DATA_BLOCK "coordinate"	// DB 22
VERSION : 0.1
  STRUCT
   CoordSaldaturaPP1 : ARRAY  [1 .. 20 ] OF //Coordinates of points
   STRUCT
    X1 : DINT ;	//X coordinate of point PP1
    Y1 : DINT ;	//Y coordinate of point PP1
    X2 : DINT ;
    Y2 : DINT ;
   END_STRUCT ;
   CoordSaldaturaPP2 : ARRAY  [1 .. 20 ] OF //Coordinates of points
   STRUCT
    X1 : DINT ;	//X coordinate of point PP2
    Y1 : DINT ;	//Y coordinate of point PP2
    X2 : DINT ;
    Y2 : DINT ;
   END_STRUCT ;
   CoordSaldaturaPP3 : ARRAY  [1 .. 20 ] OF //Coordinates of points
   STRUCT
    X1 : DINT ;	//X coordinate of point PP3
    Y1 : DINT ;	//Y coordinate of point PP3
    X2 : DINT ;
    Y2 : DINT ;
   END_STRUCT ;
   CoordSaldaturaPP4 : ARRAY  [1 .. 20 ] OF //Coordinates of points
   STRUCT
    X1 : DINT ;	//X coordinate of point PP4
    Y1 : DINT ;	//Y coordinate of point PP4
    X2 : DINT ;
    Y2 : DINT ;
   END_STRUCT ;
   CoordSaldaturaPP5 : ARRAY  [1 .. 20 ] OF //Coordinates of points
   STRUCT
    X1 : DINT ;	//X coordinate of point PP5
    Y1 : DINT ;	//Y coordinate of point PP5
    X2 : DINT ;
    Y2 : DINT ;
   END_STRUCT ;
   CoordSaldaturaPP6 : ARRAY  [1 .. 20 ] OF STRUCT
    X1 : DINT ;
    Y1 : DINT ;
    X2 : DINT ;
    Y2 : DINT ;
   END_STRUCT ;
   CoordSaldaturaPP7 : ARRAY  [1 .. 20 ] OF STRUCT
    X1 : DINT ;
    Y1 : DINT ;
    X2 : DINT ;
    Y2 : DINT ;
   END_STRUCT ;
   CoordSaldaturaPP8 : ARRAY  [1 .. 20 ] OF STRUCT
    X1 : DINT ;
    Y1 : DINT ;
    X2 : DINT ;
    Y2 : DINT ;
   END_STRUCT ;
   CoordSaldaturaPP9 : ARRAY  [1 .. 20 ] OF STRUCT
    X1 : DINT ;
    Y1 : DINT ;
    X2 : DINT ;
    Y2 : DINT ;
   END_STRUCT ;
   CoordSaldaturaPP10 : ARRAY  [1 .. 20 ] OF STRUCT
    X1 : DINT ;
    Y1 : DINT ;
    X2 : DINT ;
    Y2 : DINT ;
   END_STRUCT ;
   CoordSaldaturaPP11 : ARRAY  [1 .. 20 ] OF STRUCT
    X1 : DINT ;
    Y1 : DINT ;
    X2 : DINT ;
    Y2 : DINT ;
   END_STRUCT ;
   CoordSaldaturaPP12 : ARRAY  [1 .. 20 ] OF STRUCT
    X1 : DINT ;
    Y1 : DINT ;
    X2 : DINT ;
    Y2 : DINT ;
   END_STRUCT ;
   CoordSaldaturaPP13 : ARRAY  [1 .. 20 ] OF STRUCT
    X1 : DINT ;
    Y1 : DINT ;
    X2 : DINT ;
    Y2 : DINT ;
   END_STRUCT ;
   CoordSaldaturaPP14 : ARRAY  [1 .. 20 ] OF STRUCT
    X1 : DINT ;
    Y1 : DINT ;
    X2 : DINT ;
    Y2 : DINT ;
   END_STRUCT ;
   CoordSaldaturaPP15 : ARRAY  [1 .. 20 ] OF STRUCT
    X1 : DINT ;
    Y1 : DINT ;
    X2 : DINT ;
    Y2 : DINT ;
   END_STRUCT ;
   CoordSaldaturaPP16 : ARRAY  [1 .. 20 ] OF STRUCT
    X1 : DINT ;
    Y1 : DINT ;
    X2 : DINT ;
    Y2 : DINT ;
   END_STRUCT ;
   CoordSaldaturaPP17 : ARRAY  [1 .. 20 ] OF STRUCT
    X1 : DINT ;
    Y1 : DINT ;
    X2 : DINT ;
    Y2 : DINT ;
   END_STRUCT ;
   CoordSaldaturaPP18 : ARRAY  [1 .. 20 ] OF STRUCT
    X1 : DINT ;
    Y1 : DINT ;
    X2 : DINT ;
    Y2 : DINT ;
   END_STRUCT ;
   CoordSaldaturaPP19 : ARRAY  [1 .. 20 ] OF STRUCT
    X1 : DINT ;
    Y1 : DINT ;
    X2 : DINT ;
    Y2 : DINT ;
   END_STRUCT ;
   CoordSaldaturaPP20 : ARRAY  [1 .. 20 ] OF STRUCT
    X1 : DINT ;
    Y1 : DINT ;
    X2 : DINT ;
    Y2 : DINT ;
   END_STRUCT ;
   CoordinateCam_PP1 : ARRAY  [1 .. 10 ] OF STRUCT
    X : DINT ;	//X coordinate of point cam PP1
    Y : DINT ;	//X coordinate of point cam PP1
   END_STRUCT ;
   CoordinateCam_PP2 : ARRAY  [1 .. 10 ] OF STRUCT
    X : DINT ;	//X coordinate of point cam PP1
    Y : DINT ;	//X coordinate of point cam PP1
   END_STRUCT ;
   CoordinateCam_PP3 : ARRAY  [1 .. 10 ] OF STRUCT
    X : DINT ;	//X coordinate of point cam PP1
    Y : DINT ;	//X coordinate of point cam PP1
   END_STRUCT ;
   CoordinateCam_PP4 : ARRAY  [1 .. 10 ] OF STRUCT
    X : DINT ;	//X coordinate of point cam PP1
    Y : DINT ;	//X coordinate of point cam PP1
   END_STRUCT ;
   CoordinateCam_PP5 : ARRAY  [1 .. 10 ] OF STRUCT
    X : DINT ;	//X coordinate of point cam PP1
    Y : DINT ;	//X coordinate of point cam PP1
   END_STRUCT ;
   CoordinateCam_PP6 : ARRAY  [1 .. 10 ] OF STRUCT
    X : DINT ;	//X coordinate of point cam PP1
    Y : DINT ;	//X coordinate of point cam PP1
   END_STRUCT ;
   CoordinateCam_PP7 : ARRAY  [1 .. 10 ] OF STRUCT
    X : DINT ;	//X coordinate of point cam PP1
    Y : DINT ;	//X coordinate of point cam PP1
   END_STRUCT ;
   CoordinateCam_PP8 : ARRAY  [1 .. 10 ] OF STRUCT
    X : DINT ;	//X coordinate of point cam PP1
    Y : DINT ;	//X coordinate of point cam PP1
   END_STRUCT ;
   CoordinateCam_PP9 : ARRAY  [1 .. 10 ] OF STRUCT
    X : DINT ;	//X coordinate of point cam PP1
    Y : DINT ;	//X coordinate of point cam PP1
   END_STRUCT ;
   CoordinateCam_PP10 : ARRAY  [1 .. 10 ] OF STRUCT
    X : DINT ;	//X coordinate of point cam PP1
    Y : DINT ;	//X coordinate of point cam PP1
   END_STRUCT ;
   CoordinateCam_PP11 : ARRAY  [1 .. 10 ] OF STRUCT
    X : DINT ;	//X coordinate of point cam PP1
    Y : DINT ;	//X coordinate of point cam PP1
   END_STRUCT ;
   CoordinateCam_PP12 : ARRAY  [1 .. 10 ] OF STRUCT
    X : DINT ;	//X coordinate of point cam PP1
    Y : DINT ;	//X coordinate of point cam PP1
   END_STRUCT ;
   CoordinateCam_PP13 : ARRAY  [1 .. 10 ] OF STRUCT
    X : DINT ;	//X coordinate of point cam PP1
    Y : DINT ;	//X coordinate of point cam PP1
   END_STRUCT ;
   CoordinateCam_PP14 : ARRAY  [1 .. 10 ] OF STRUCT
    X : DINT ;	//X coordinate of point cam PP1
    Y : DINT ;	//X coordinate of point cam PP1
   END_STRUCT ;
   CoordinateCam_PP15 : ARRAY  [1 .. 10 ] OF STRUCT
    X : DINT ;	//X coordinate of point cam PP1
    Y : DINT ;	//X coordinate of point cam PP1
   END_STRUCT ;
   CoordinateCam_PP16 : ARRAY  [1 .. 10 ] OF STRUCT
    X : DINT ;	//X coordinate of point cam PP1
    Y : DINT ;	//X coordinate of point cam PP1
   END_STRUCT ;
   CoordinateCam_PP17 : ARRAY  [1 .. 10 ] OF STRUCT
    X : DINT ;	//X coordinate of point cam PP1
    Y : DINT ;	//X coordinate of point cam PP1
   END_STRUCT ;
   CoordinateCam_PP18 : ARRAY  [1 .. 10 ] OF STRUCT
    X : DINT ;	//X coordinate of point cam PP1
    Y : DINT ;	//X coordinate of point cam PP1
   END_STRUCT ;
   CoordinateCam_PP19 : ARRAY  [1 .. 10 ] OF STRUCT
    X : DINT ;	//X coordinate of point cam PP1
    Y : DINT ;	//X coordinate of point cam PP1
   END_STRUCT ;
   CoordinateCam_PP20 : ARRAY  [1 .. 10 ] OF STRUCT
    X : DINT ;	//X coordinate of point cam PP1
    Y : DINT ;	//X coordinate of point cam PP1
   END_STRUCT ;
   NumeroSaldaturePP1 : INT ;
   NumeroSaldaturePP2 : INT ;
   NumeroSaldaturePP3 : INT ;
   NumeroSaldaturePP4 : INT ;
   NumeroSaldaturePP5 : INT ;
   NumeroSaldaturePP6 : INT ;
   NumeroSaldaturePP7 : INT ;
   NumeroSaldaturePP8 : INT ;
   NumeroSaldaturePP9 : INT ;
   NumeroSaldaturePP10 : INT ;
   NumeroSaldaturePP11 : INT ;
   NumeroSaldaturePP12 : INT ;
   NumeroSaldaturePP13 : INT ;
   NumeroSaldaturePP14 : INT ;
   NumeroSaldaturePP15 : INT ;
   NumeroSaldaturePP16 : INT ;
   NumeroSaldaturePP17 : INT ;
   NumeroSaldaturePP18 : INT ;
   NumeroSaldaturePP19 : INT ;
   NumeroSaldaturePP20 : INT ;
   TimeWeldingPP1 : ARRAY  [1 .. 20 ] OF STRUCT
    Tempo : S5TIME  := S5T#1S;
   END_STRUCT ;
   TimeWeldingPP2 : ARRAY  [1 .. 20 ] OF STRUCT
    Tempo : S5TIME  := S5T#1S;
   END_STRUCT ;
   TimeWeldingPP3 : ARRAY  [1 .. 20 ] OF STRUCT
    Tempo : S5TIME  := S5T#1S;
   END_STRUCT ;
   TimeWeldingPP4 : ARRAY  [1 .. 20 ] OF STRUCT
    Tempo : S5TIME  := S5T#1S;
   END_STRUCT ;
   TimeWeldingPP5 : ARRAY  [1 .. 20 ] OF STRUCT
    Tempo : S5TIME  := S5T#1S;
   END_STRUCT ;
   TimeWeldingPP6 : ARRAY  [1 .. 20 ] OF STRUCT
    Tempo : S5TIME  := S5T#1S;
   END_STRUCT ;
   TimeWeldingPP7 : ARRAY  [1 .. 20 ] OF STRUCT
    Tempo : S5TIME  := S5T#1S;
   END_STRUCT ;
   TimeWeldingPP8 : ARRAY  [1 .. 20 ] OF STRUCT
    Tempo : S5TIME  := S5T#1S;
   END_STRUCT ;
   TimeWeldingPP9 : ARRAY  [1 .. 20 ] OF STRUCT
    Tempo : S5TIME  := S5T#1S;
   END_STRUCT ;
   TimeWeldingPP10 : ARRAY  [1 .. 20 ] OF STRUCT
    Tempo : S5TIME  := S5T#1S;
   END_STRUCT ;
   TimeWeldingPP11 : ARRAY  [1 .. 20 ] OF STRUCT
    Tempo : S5TIME  := S5T#1S;
   END_STRUCT ;
   TimeWeldingPP12 : ARRAY  [1 .. 20 ] OF STRUCT
    Tempo : S5TIME  := S5T#1S;
   END_STRUCT ;
   TimeWeldingPP13 : ARRAY  [1 .. 20 ] OF STRUCT
    Tempo : S5TIME  := S5T#1S;
   END_STRUCT ;
   TimeWeldingPP14 : ARRAY  [1 .. 20 ] OF STRUCT
    Tempo : S5TIME  := S5T#1S;
   END_STRUCT ;
   TimeWeldingPP15 : ARRAY  [1 .. 20 ] OF STRUCT
    Tempo : S5TIME  := S5T#1S;
   END_STRUCT ;
   TimeWeldingPP16 : ARRAY  [1 .. 20 ] OF STRUCT
    Tempo : S5TIME  := S5T#1S;
   END_STRUCT ;
   TimeWeldingPP17 : ARRAY  [1 .. 20 ] OF STRUCT
    Tempo : S5TIME  := S5T#1S;
   END_STRUCT ;
   TimeWeldingPP18 : ARRAY  [1 .. 20 ] OF STRUCT
    Tempo : S5TIME  := S5T#1S;
   END_STRUCT ;
   TimeWeldingPP19 : ARRAY  [1 .. 20 ] OF STRUCT
    Tempo : S5TIME  := S5T#1S;
   END_STRUCT ;
   TimeWeldingPP20 : ARRAY  [1 .. 20 ] OF STRUCT
    Tempo : S5TIME  := S5T#1S;
   END_STRUCT ;
  END_STRUCT ;	
BEGIN
   CoordSaldaturaPP1[1].X1 := L#-60530;
   CoordSaldaturaPP1[1].Y1 := L#-172340;
   CoordSaldaturaPP1[1].X2 := L#-60530;
   CoordSaldaturaPP1[1].Y2 := L#-172340;
   CoordSaldaturaPP1[2].X1 := L#-46530;
   CoordSaldaturaPP1[2].Y1 := L#-162870;
   CoordSaldaturaPP1[2].X2 := L#-46530;
   CoordSaldaturaPP1[2].Y2 := L#-162870;
   CoordSaldaturaPP1[3].X1 := L#-29630;
   CoordSaldaturaPP1[3].Y1 := L#-163440;
   CoordSaldaturaPP1[3].X2 := L#-29630;
   CoordSaldaturaPP1[3].Y2 := L#-163440;
   CoordSaldaturaPP1[4].X1 := L#-16300;
   CoordSaldaturaPP1[4].Y1 := L#-173820;
   CoordSaldaturaPP1[4].X2 := L#-16300;
   CoordSaldaturaPP1[4].Y2 := L#-173820;
   CoordSaldaturaPP1[5].X1 := L#-11620;
   CoordSaldaturaPP1[5].Y1 := L#-190070;
   CoordSaldaturaPP1[5].X2 := L#-11620;
   CoordSaldaturaPP1[5].Y2 := L#-190070;
   CoordSaldaturaPP1[6].X1 := L#-17370;
   CoordSaldaturaPP1[6].Y1 := L#-205960;
   CoordSaldaturaPP1[6].X2 := L#-17370;
   CoordSaldaturaPP1[6].Y2 := L#-205960;
   CoordSaldaturaPP1[7].X1 := L#-31370;
   CoordSaldaturaPP1[7].Y1 := L#-215430;
   CoordSaldaturaPP1[7].X2 := L#-31370;
   CoordSaldaturaPP1[7].Y2 := L#-215430;
   CoordSaldaturaPP1[8].X1 := L#-48270;
   CoordSaldaturaPP1[8].Y1 := L#-214860;
   CoordSaldaturaPP1[8].X2 := L#-48270;
   CoordSaldaturaPP1[8].Y2 := L#-214860;
   CoordSaldaturaPP1[9].X1 := L#-61600;
   CoordSaldaturaPP1[9].Y1 := L#-204480;
   CoordSaldaturaPP1[9].X2 := L#-61600;
   CoordSaldaturaPP1[9].Y2 := L#-204480;
   CoordSaldaturaPP1[10].X1 := L#-66280;
   CoordSaldaturaPP1[10].Y1 := L#-188230;
   CoordSaldaturaPP1[10].X2 := L#-66280;
   CoordSaldaturaPP1[10].Y2 := L#-188230;
   CoordSaldaturaPP6[1].X1 := L#-24431;
   CoordSaldaturaPP6[1].Y1 := L#-211667;
   CoordSaldaturaPP6[1].X2 := L#-24468;
   CoordSaldaturaPP6[1].Y2 := L#-211634;
   CoordSaldaturaPP6[2].X1 := L#-13011;
   CoordSaldaturaPP6[2].Y1 := L#-199436;
   CoordSaldaturaPP6[2].X2 := L#-12856;
   CoordSaldaturaPP6[2].Y2 := L#-199488;
   CoordSaldaturaPP6[3].X1 := L#-9745;
   CoordSaldaturaPP6[3].Y1 := L#-183598;
   CoordSaldaturaPP6[3].X2 := L#-9756;
   CoordSaldaturaPP6[3].Y2 := L#-183663;
   CoordSaldaturaPP6[4].X1 := L#-16203;
   CoordSaldaturaPP6[4].Y1 := L#-168150;
   CoordSaldaturaPP6[4].X2 := L#-16141;
   CoordSaldaturaPP6[4].Y2 := L#-168156;
   CoordSaldaturaPP6[5].X1 := L#-29434;
   CoordSaldaturaPP6[5].Y1 := L#-158429;
   CoordSaldaturaPP6[5].X2 := L#-29472;
   CoordSaldaturaPP6[5].Y2 := L#-158489;
   CoordSaldaturaPP6[6].X1 := L#-46262;
   CoordSaldaturaPP6[6].Y1 := L#-157658;
   CoordSaldaturaPP6[6].X2 := L#-46155;
   CoordSaldaturaPP6[6].Y2 := L#-157716;
   CoordSaldaturaPP6[7].X1 := L#-60740;
   CoordSaldaturaPP6[7].Y1 := L#-166127;
   CoordSaldaturaPP6[7].X2 := L#-60564;
   CoordSaldaturaPP6[7].Y2 := L#-166296;
   CoordSaldaturaPP6[8].X1 := L#-68335;
   CoordSaldaturaPP6[8].Y1 := L#-180765;
   CoordSaldaturaPP6[8].X2 := L#-68026;
   CoordSaldaturaPP6[8].Y2 := L#-180787;
   CoordSaldaturaPP6[9].X1 := L#-66468;
   CoordSaldaturaPP6[9].Y1 := L#-197254;
   CoordSaldaturaPP6[9].X2 := L#-66217;
   CoordSaldaturaPP6[9].Y2 := L#-197398;
   CoordSaldaturaPP6[10].X1 := L#-56162;
   CoordSaldaturaPP6[10].Y1 := L#-210332;
   CoordSaldaturaPP6[10].X2 := L#-56200;
   CoordSaldaturaPP6[10].Y2 := L#-210331;
   CoordSaldaturaPP6[11].X1 := L#-40981;
   CoordSaldaturaPP6[11].Y1 := L#-215911;
   CoordSaldaturaPP6[11].X2 := L#-40587;
   CoordSaldaturaPP6[11].Y2 := L#-215681;
   CoordSaldaturaPP11[1].X1 := L#-24431;
   CoordSaldaturaPP11[1].Y1 := L#-211667;
   CoordSaldaturaPP11[1].X2 := L#-24468;
   CoordSaldaturaPP11[1].Y2 := L#-211634;
   CoordSaldaturaPP11[2].X1 := L#-13011;
   CoordSaldaturaPP11[2].Y1 := L#-199436;
   CoordSaldaturaPP11[2].X2 := L#-12856;
   CoordSaldaturaPP11[2].Y2 := L#-199488;
   CoordSaldaturaPP11[3].X1 := L#-9745;
   CoordSaldaturaPP11[3].Y1 := L#-183598;
   CoordSaldaturaPP11[3].X2 := L#-9786;
   CoordSaldaturaPP11[3].Y2 := L#-183663;
   CoordSaldaturaPP11[4].X1 := L#-16203;
   CoordSaldaturaPP11[4].Y1 := L#-168150;
   CoordSaldaturaPP11[4].X2 := L#-16141;
   CoordSaldaturaPP11[4].Y2 := L#-168156;
   CoordSaldaturaPP11[5].X1 := L#-29434;
   CoordSaldaturaPP11[5].Y1 := L#-158429;
   CoordSaldaturaPP11[5].X2 := L#-29472;
   CoordSaldaturaPP11[5].Y2 := L#-158489;
   CoordSaldaturaPP11[6].X1 := L#-46262;
   CoordSaldaturaPP11[6].Y1 := L#-157658;
   CoordSaldaturaPP11[6].X2 := L#-46155;
   CoordSaldaturaPP11[6].Y2 := L#-157716;
   CoordSaldaturaPP11[7].X1 := L#-60740;
   CoordSaldaturaPP11[7].Y1 := L#-166127;
   CoordSaldaturaPP11[7].X2 := L#-60564;
   CoordSaldaturaPP11[7].Y2 := L#-166296;
   CoordSaldaturaPP11[8].X1 := L#-68335;
   CoordSaldaturaPP11[8].Y1 := L#-180765;
   CoordSaldaturaPP11[8].X2 := L#-68026;
   CoordSaldaturaPP11[8].Y2 := L#-180787;
   CoordSaldaturaPP11[9].X1 := L#-66468;
   CoordSaldaturaPP11[9].Y1 := L#-197254;
   CoordSaldaturaPP11[9].X2 := L#-66217;
   CoordSaldaturaPP11[9].Y2 := L#-197398;
   CoordSaldaturaPP11[10].X1 := L#-56162;
   CoordSaldaturaPP11[10].Y1 := L#-210332;
   CoordSaldaturaPP11[10].X2 := L#-56200;
   CoordSaldaturaPP11[10].Y2 := L#-210331;
   CoordSaldaturaPP11[11].X1 := L#-40981;
   CoordSaldaturaPP11[11].Y1 := L#-215911;
   CoordSaldaturaPP11[11].X2 := L#-40587;
   CoordSaldaturaPP11[11].Y2 := L#-215681;
   CoordinateCam_PP1[1].X := L#7915;
   CoordinateCam_PP1[1].Y := L#-68282;
   NumeroSaldaturePP1 := 10;
   TimeWeldingPP1[1].Tempo := S5T#1S;
   TimeWeldingPP1[2].Tempo := S5T#2S;
   TimeWeldingPP1[3].Tempo := S5T#1S;
   TimeWeldingPP1[4].Tempo := S5T#1S;
   TimeWeldingPP1[5].Tempo := S5T#1S;
   TimeWeldingPP1[6].Tempo := S5T#1S;
   TimeWeldingPP1[7].Tempo := S5T#1S;
   TimeWeldingPP1[8].Tempo := S5T#1S;
   TimeWeldingPP1[9].Tempo := S5T#1S;
   TimeWeldingPP1[10].Tempo := S5T#1S;
   TimeWeldingPP1[11].Tempo := S5T#1S;
   TimeWeldingPP1[12].Tempo := S5T#1S;
   TimeWeldingPP1[13].Tempo := S5T#1S;
   TimeWeldingPP1[14].Tempo := S5T#1S;
   TimeWeldingPP1[15].Tempo := S5T#1S;
   TimeWeldingPP1[16].Tempo := S5T#1S;
   TimeWeldingPP1[17].Tempo := S5T#1S;
   TimeWeldingPP1[18].Tempo := S5T#1S;
   TimeWeldingPP1[19].Tempo := S5T#1S;
   TimeWeldingPP1[20].Tempo := S5T#1S;
   TimeWeldingPP2[1].Tempo := S5T#1S;
   TimeWeldingPP2[2].Tempo := S5T#1S;
   TimeWeldingPP2[3].Tempo := S5T#1S;
   TimeWeldingPP2[4].Tempo := S5T#1S;
   TimeWeldingPP2[5].Tempo := S5T#1S;
   TimeWeldingPP2[6].Tempo := S5T#1S;
   TimeWeldingPP2[7].Tempo := S5T#1S;
   TimeWeldingPP2[8].Tempo := S5T#1S;
   TimeWeldingPP2[9].Tempo := S5T#1S;
   TimeWeldingPP2[10].Tempo := S5T#1S;
   TimeWeldingPP2[11].Tempo := S5T#1S;
   TimeWeldingPP2[12].Tempo := S5T#1S;
   TimeWeldingPP2[13].Tempo := S5T#1S;
   TimeWeldingPP2[14].Tempo := S5T#1S;
   TimeWeldingPP2[15].Tempo := S5T#1S;
   TimeWeldingPP2[16].Tempo := S5T#1S;
   TimeWeldingPP2[17].Tempo := S5T#1S;
   TimeWeldingPP2[18].Tempo := S5T#1S;
   TimeWeldingPP2[19].Tempo := S5T#1S;
   TimeWeldingPP2[20].Tempo := S5T#1S;
   TimeWeldingPP3[1].Tempo := S5T#1S;
   TimeWeldingPP3[2].Tempo := S5T#1S;
   TimeWeldingPP3[3].Tempo := S5T#1S;
   TimeWeldingPP3[4].Tempo := S5T#1S;
   TimeWeldingPP3[5].Tempo := S5T#1S;
   TimeWeldingPP3[6].Tempo := S5T#1S;
   TimeWeldingPP3[7].Tempo := S5T#1S;
   TimeWeldingPP3[8].Tempo := S5T#1S;
   TimeWeldingPP3[9].Tempo := S5T#1S;
   TimeWeldingPP3[10].Tempo := S5T#1S;
   TimeWeldingPP3[11].Tempo := S5T#1S;
   TimeWeldingPP3[12].Tempo := S5T#1S;
   TimeWeldingPP3[13].Tempo := S5T#1S;
   TimeWeldingPP3[14].Tempo := S5T#1S;
   TimeWeldingPP3[15].Tempo := S5T#1S;
   TimeWeldingPP3[16].Tempo := S5T#1S;
   TimeWeldingPP3[17].Tempo := S5T#1S;
   TimeWeldingPP3[18].Tempo := S5T#1S;
   TimeWeldingPP3[19].Tempo := S5T#1S;
   TimeWeldingPP3[20].Tempo := S5T#1S;
   TimeWeldingPP4[1].Tempo := S5T#1S;
   TimeWeldingPP4[2].Tempo := S5T#1S;
   TimeWeldingPP4[3].Tempo := S5T#1S;
   TimeWeldingPP4[4].Tempo := S5T#1S;
   TimeWeldingPP4[5].Tempo := S5T#1S;
   TimeWeldingPP4[6].Tempo := S5T#1S;
   TimeWeldingPP4[7].Tempo := S5T#1S;
   TimeWeldingPP4[8].Tempo := S5T#1S;
   TimeWeldingPP4[9].Tempo := S5T#1S;
   TimeWeldingPP4[10].Tempo := S5T#1S;
   TimeWeldingPP4[11].Tempo := S5T#1S;
   TimeWeldingPP4[12].Tempo := S5T#1S;
   TimeWeldingPP4[13].Tempo := S5T#1S;
   TimeWeldingPP4[14].Tempo := S5T#1S;
   TimeWeldingPP4[15].Tempo := S5T#1S;
   TimeWeldingPP4[16].Tempo := S5T#1S;
   TimeWeldingPP4[17].Tempo := S5T#1S;
   TimeWeldingPP4[18].Tempo := S5T#1S;
   TimeWeldingPP4[19].Tempo := S5T#1S;
   TimeWeldingPP4[20].Tempo := S5T#1S;
   TimeWeldingPP5[1].Tempo := S5T#1S;
   TimeWeldingPP5[2].Tempo := S5T#1S;
   TimeWeldingPP5[3].Tempo := S5T#1S;
   TimeWeldingPP5[4].Tempo := S5T#1S;
   TimeWeldingPP5[5].Tempo := S5T#1S;
   TimeWeldingPP5[6].Tempo := S5T#1S;
   TimeWeldingPP5[7].Tempo := S5T#1S;
   TimeWeldingPP5[8].Tempo := S5T#1S;
   TimeWeldingPP5[9].Tempo := S5T#1S;
   TimeWeldingPP5[10].Tempo := S5T#1S;
   TimeWeldingPP5[11].Tempo := S5T#1S;
   TimeWeldingPP5[12].Tempo := S5T#1S;
   TimeWeldingPP5[13].Tempo := S5T#1S;
   TimeWeldingPP5[14].Tempo := S5T#1S;
   TimeWeldingPP5[15].Tempo := S5T#1S;
   TimeWeldingPP5[16].Tempo := S5T#1S;
   TimeWeldingPP5[17].Tempo := S5T#1S;
   TimeWeldingPP5[18].Tempo := S5T#1S;
   TimeWeldingPP5[19].Tempo := S5T#1S;
   TimeWeldingPP5[20].Tempo := S5T#1S;
   TimeWeldingPP6[1].Tempo := S5T#1S;
   TimeWeldingPP6[2].Tempo := S5T#1S;
   TimeWeldingPP6[3].Tempo := S5T#1S;
   TimeWeldingPP6[4].Tempo := S5T#1S;
   TimeWeldingPP6[5].Tempo := S5T#1S;
   TimeWeldingPP6[6].Tempo := S5T#1S;
   TimeWeldingPP6[7].Tempo := S5T#1S;
   TimeWeldingPP6[8].Tempo := S5T#1S;
   TimeWeldingPP6[9].Tempo := S5T#1S;
   TimeWeldingPP6[10].Tempo := S5T#1S;
   TimeWeldingPP6[11].Tempo := S5T#1S;
   TimeWeldingPP6[12].Tempo := S5T#1S;
   TimeWeldingPP6[13].Tempo := S5T#1S;
   TimeWeldingPP6[14].Tempo := S5T#1S;
   TimeWeldingPP6[15].Tempo := S5T#1S;
   TimeWeldingPP6[16].Tempo := S5T#1S;
   TimeWeldingPP6[17].Tempo := S5T#1S;
   TimeWeldingPP6[18].Tempo := S5T#1S;
   TimeWeldingPP6[19].Tempo := S5T#1S;
   TimeWeldingPP6[20].Tempo := S5T#1S;
   TimeWeldingPP7[1].Tempo := S5T#1S;
   TimeWeldingPP7[2].Tempo := S5T#1S;
   TimeWeldingPP7[3].Tempo := S5T#1S;
   TimeWeldingPP7[4].Tempo := S5T#1S;
   TimeWeldingPP7[5].Tempo := S5T#1S;
   TimeWeldingPP7[6].Tempo := S5T#1S;
   TimeWeldingPP7[7].Tempo := S5T#1S;
   TimeWeldingPP7[8].Tempo := S5T#1S;
   TimeWeldingPP7[9].Tempo := S5T#1S;
   TimeWeldingPP7[10].Tempo := S5T#1S;
   TimeWeldingPP7[11].Tempo := S5T#1S;
   TimeWeldingPP7[12].Tempo := S5T#1S;
   TimeWeldingPP7[13].Tempo := S5T#1S;
   TimeWeldingPP7[14].Tempo := S5T#1S;
   TimeWeldingPP7[15].Tempo := S5T#1S;
   TimeWeldingPP7[16].Tempo := S5T#1S;
   TimeWeldingPP7[17].Tempo := S5T#1S;
   TimeWeldingPP7[18].Tempo := S5T#1S;
   TimeWeldingPP7[19].Tempo := S5T#1S;
   TimeWeldingPP7[20].Tempo := S5T#1S;
   TimeWeldingPP8[1].Tempo := S5T#1S;
   TimeWeldingPP8[2].Tempo := S5T#1S;
   TimeWeldingPP8[3].Tempo := S5T#1S;
   TimeWeldingPP8[4].Tempo := S5T#1S;
   TimeWeldingPP8[5].Tempo := S5T#1S;
   TimeWeldingPP8[6].Tempo := S5T#1S;
   TimeWeldingPP8[7].Tempo := S5T#1S;
   TimeWeldingPP8[8].Tempo := S5T#1S;
   TimeWeldingPP8[9].Tempo := S5T#1S;
   TimeWeldingPP8[10].Tempo := S5T#1S;
   TimeWeldingPP8[11].Tempo := S5T#1S;
   TimeWeldingPP8[12].Tempo := S5T#1S;
   TimeWeldingPP8[13].Tempo := S5T#1S;
   TimeWeldingPP8[14].Tempo := S5T#1S;
   TimeWeldingPP8[15].Tempo := S5T#1S;
   TimeWeldingPP8[16].Tempo := S5T#1S;
   TimeWeldingPP8[17].Tempo := S5T#1S;
   TimeWeldingPP8[18].Tempo := S5T#1S;
   TimeWeldingPP8[19].Tempo := S5T#1S;
   TimeWeldingPP8[20].Tempo := S5T#1S;
   TimeWeldingPP9[1].Tempo := S5T#1S;
   TimeWeldingPP9[2].Tempo := S5T#1S;
   TimeWeldingPP9[3].Tempo := S5T#1S;
   TimeWeldingPP9[4].Tempo := S5T#1S;
   TimeWeldingPP9[5].Tempo := S5T#1S;
   TimeWeldingPP9[6].Tempo := S5T#1S;
   TimeWeldingPP9[7].Tempo := S5T#1S;
   TimeWeldingPP9[8].Tempo := S5T#1S;
   TimeWeldingPP9[9].Tempo := S5T#1S;
   TimeWeldingPP9[10].Tempo := S5T#1S;
   TimeWeldingPP9[11].Tempo := S5T#1S;
   TimeWeldingPP9[12].Tempo := S5T#1S;
   TimeWeldingPP9[13].Tempo := S5T#1S;
   TimeWeldingPP9[14].Tempo := S5T#1S;
   TimeWeldingPP9[15].Tempo := S5T#1S;
   TimeWeldingPP9[16].Tempo := S5T#1S;
   TimeWeldingPP9[17].Tempo := S5T#1S;
   TimeWeldingPP9[18].Tempo := S5T#1S;
   TimeWeldingPP9[19].Tempo := S5T#1S;
   TimeWeldingPP9[20].Tempo := S5T#1S;
   TimeWeldingPP10[1].Tempo := S5T#1S;
   TimeWeldingPP10[2].Tempo := S5T#1S;
   TimeWeldingPP10[3].Tempo := S5T#1S;
   TimeWeldingPP10[4].Tempo := S5T#1S;
   TimeWeldingPP10[5].Tempo := S5T#1S;
   TimeWeldingPP10[6].Tempo := S5T#1S;
   TimeWeldingPP10[7].Tempo := S5T#1S;
   TimeWeldingPP10[8].Tempo := S5T#1S;
   TimeWeldingPP10[9].Tempo := S5T#1S;
   TimeWeldingPP10[10].Tempo := S5T#1S;
   TimeWeldingPP10[11].Tempo := S5T#1S;
   TimeWeldingPP10[12].Tempo := S5T#1S;
   TimeWeldingPP10[13].Tempo := S5T#1S;
   TimeWeldingPP10[14].Tempo := S5T#1S;
   TimeWeldingPP10[15].Tempo := S5T#1S;
   TimeWeldingPP10[16].Tempo := S5T#1S;
   TimeWeldingPP10[17].Tempo := S5T#1S;
   TimeWeldingPP10[18].Tempo := S5T#1S;
   TimeWeldingPP10[19].Tempo := S5T#1S;
   TimeWeldingPP10[20].Tempo := S5T#1S;
   TimeWeldingPP11[1].Tempo := S5T#1S700MS;
   TimeWeldingPP11[2].Tempo := S5T#1S;
   TimeWeldingPP11[3].Tempo := S5T#1S;
   TimeWeldingPP11[4].Tempo := S5T#1S;
   TimeWeldingPP11[5].Tempo := S5T#1S;
   TimeWeldingPP11[6].Tempo := S5T#1S;
   TimeWeldingPP11[7].Tempo := S5T#1S;
   TimeWeldingPP11[8].Tempo := S5T#1S;
   TimeWeldingPP11[9].Tempo := S5T#1S;
   TimeWeldingPP11[10].Tempo := S5T#1S;
   TimeWeldingPP11[11].Tempo := S5T#1S;
   TimeWeldingPP11[12].Tempo := S5T#1S;
   TimeWeldingPP11[13].Tempo := S5T#1S;
   TimeWeldingPP11[14].Tempo := S5T#1S;
   TimeWeldingPP11[15].Tempo := S5T#1S;
   TimeWeldingPP11[16].Tempo := S5T#1S;
   TimeWeldingPP11[17].Tempo := S5T#1S;
   TimeWeldingPP11[18].Tempo := S5T#1S;
   TimeWeldingPP11[19].Tempo := S5T#1S;
   TimeWeldingPP11[20].Tempo := S5T#1S;
   TimeWeldingPP12[1].Tempo := S5T#1S;
   TimeWeldingPP12[2].Tempo := S5T#1S;
   TimeWeldingPP12[3].Tempo := S5T#1S;
   TimeWeldingPP12[4].Tempo := S5T#1S;
   TimeWeldingPP12[5].Tempo := S5T#1S;
   TimeWeldingPP12[6].Tempo := S5T#1S;
   TimeWeldingPP12[7].Tempo := S5T#1S;
   TimeWeldingPP12[8].Tempo := S5T#1S;
   TimeWeldingPP12[9].Tempo := S5T#1S;
   TimeWeldingPP12[10].Tempo := S5T#1S;
   TimeWeldingPP12[11].Tempo := S5T#1S;
   TimeWeldingPP12[12].Tempo := S5T#1S;
   TimeWeldingPP12[13].Tempo := S5T#1S;
   TimeWeldingPP12[14].Tempo := S5T#1S;
   TimeWeldingPP12[15].Tempo := S5T#1S;
   TimeWeldingPP12[16].Tempo := S5T#1S;
   TimeWeldingPP12[17].Tempo := S5T#1S;
   TimeWeldingPP12[18].Tempo := S5T#1S;
   TimeWeldingPP12[19].Tempo := S5T#1S;
   TimeWeldingPP12[20].Tempo := S5T#1S;
   TimeWeldingPP13[1].Tempo := S5T#1S;
   TimeWeldingPP13[2].Tempo := S5T#1S;
   TimeWeldingPP13[3].Tempo := S5T#1S;
   TimeWeldingPP13[4].Tempo := S5T#1S;
   TimeWeldingPP13[5].Tempo := S5T#1S;
   TimeWeldingPP13[6].Tempo := S5T#1S;
   TimeWeldingPP13[7].Tempo := S5T#1S;
   TimeWeldingPP13[8].Tempo := S5T#1S;
   TimeWeldingPP13[9].Tempo := S5T#1S;
   TimeWeldingPP13[10].Tempo := S5T#1S;
   TimeWeldingPP13[11].Tempo := S5T#1S;
   TimeWeldingPP13[12].Tempo := S5T#1S;
   TimeWeldingPP13[13].Tempo := S5T#1S;
   TimeWeldingPP13[14].Tempo := S5T#1S;
   TimeWeldingPP13[15].Tempo := S5T#1S;
   TimeWeldingPP13[16].Tempo := S5T#1S;
   TimeWeldingPP13[17].Tempo := S5T#1S;
   TimeWeldingPP13[18].Tempo := S5T#1S;
   TimeWeldingPP13[19].Tempo := S5T#1S;
   TimeWeldingPP13[20].Tempo := S5T#1S;
   TimeWeldingPP14[1].Tempo := S5T#1S;
   TimeWeldingPP14[2].Tempo := S5T#1S;
   TimeWeldingPP14[3].Tempo := S5T#1S;
   TimeWeldingPP14[4].Tempo := S5T#1S;
   TimeWeldingPP14[5].Tempo := S5T#1S;
   TimeWeldingPP14[6].Tempo := S5T#1S;
   TimeWeldingPP14[7].Tempo := S5T#1S;
   TimeWeldingPP14[8].Tempo := S5T#1S;
   TimeWeldingPP14[9].Tempo := S5T#1S;
   TimeWeldingPP14[10].Tempo := S5T#1S;
   TimeWeldingPP14[11].Tempo := S5T#1S;
   TimeWeldingPP14[12].Tempo := S5T#1S;
   TimeWeldingPP14[13].Tempo := S5T#1S;
   TimeWeldingPP14[14].Tempo := S5T#1S;
   TimeWeldingPP14[15].Tempo := S5T#1S;
   TimeWeldingPP14[16].Tempo := S5T#1S;
   TimeWeldingPP14[17].Tempo := S5T#1S;
   TimeWeldingPP14[18].Tempo := S5T#1S;
   TimeWeldingPP14[19].Tempo := S5T#1S;
   TimeWeldingPP14[20].Tempo := S5T#1S;
   TimeWeldingPP15[1].Tempo := S5T#1S;
   TimeWeldingPP15[2].Tempo := S5T#1S;
   TimeWeldingPP15[3].Tempo := S5T#1S;
   TimeWeldingPP15[4].Tempo := S5T#1S;
   TimeWeldingPP15[5].Tempo := S5T#1S;
   TimeWeldingPP15[6].Tempo := S5T#1S;
   TimeWeldingPP15[7].Tempo := S5T#1S;
   TimeWeldingPP15[8].Tempo := S5T#1S;
   TimeWeldingPP15[9].Tempo := S5T#1S;
   TimeWeldingPP15[10].Tempo := S5T#1S;
   TimeWeldingPP15[11].Tempo := S5T#1S;
   TimeWeldingPP15[12].Tempo := S5T#1S;
   TimeWeldingPP15[13].Tempo := S5T#1S;
   TimeWeldingPP15[14].Tempo := S5T#1S;
   TimeWeldingPP15[15].Tempo := S5T#1S;
   TimeWeldingPP15[16].Tempo := S5T#1S;
   TimeWeldingPP15[17].Tempo := S5T#1S;
   TimeWeldingPP15[18].Tempo := S5T#1S;
   TimeWeldingPP15[19].Tempo := S5T#1S;
   TimeWeldingPP15[20].Tempo := S5T#1S;
   TimeWeldingPP16[1].Tempo := S5T#1S;
   TimeWeldingPP16[2].Tempo := S5T#1S;
   TimeWeldingPP16[3].Tempo := S5T#1S;
   TimeWeldingPP16[4].Tempo := S5T#1S;
   TimeWeldingPP16[5].Tempo := S5T#1S;
   TimeWeldingPP16[6].Tempo := S5T#1S;
   TimeWeldingPP16[7].Tempo := S5T#1S;
   TimeWeldingPP16[8].Tempo := S5T#1S;
   TimeWeldingPP16[9].Tempo := S5T#1S;
   TimeWeldingPP16[10].Tempo := S5T#1S;
   TimeWeldingPP16[11].Tempo := S5T#1S;
   TimeWeldingPP16[12].Tempo := S5T#1S;
   TimeWeldingPP16[13].Tempo := S5T#1S;
   TimeWeldingPP16[14].Tempo := S5T#1S;
   TimeWeldingPP16[15].Tempo := S5T#1S;
   TimeWeldingPP16[16].Tempo := S5T#1S;
   TimeWeldingPP16[17].Tempo := S5T#1S;
   TimeWeldingPP16[18].Tempo := S5T#1S;
   TimeWeldingPP16[19].Tempo := S5T#1S;
   TimeWeldingPP16[20].Tempo := S5T#1S;
   TimeWeldingPP17[1].Tempo := S5T#1S;
   TimeWeldingPP17[2].Tempo := S5T#1S;
   TimeWeldingPP17[3].Tempo := S5T#1S;
   TimeWeldingPP17[4].Tempo := S5T#1S;
   TimeWeldingPP17[5].Tempo := S5T#1S;
   TimeWeldingPP17[6].Tempo := S5T#1S;
   TimeWeldingPP17[7].Tempo := S5T#1S;
   TimeWeldingPP17[8].Tempo := S5T#1S;
   TimeWeldingPP17[9].Tempo := S5T#1S;
   TimeWeldingPP17[10].Tempo := S5T#1S;
   TimeWeldingPP17[11].Tempo := S5T#1S;
   TimeWeldingPP17[12].Tempo := S5T#1S;
   TimeWeldingPP17[13].Tempo := S5T#1S;
   TimeWeldingPP17[14].Tempo := S5T#1S;
   TimeWeldingPP17[15].Tempo := S5T#1S;
   TimeWeldingPP17[16].Tempo := S5T#1S;
   TimeWeldingPP17[17].Tempo := S5T#1S;
   TimeWeldingPP17[18].Tempo := S5T#1S;
   TimeWeldingPP17[19].Tempo := S5T#1S;
   TimeWeldingPP17[20].Tempo := S5T#1S;
   TimeWeldingPP18[1].Tempo := S5T#1S;
   TimeWeldingPP18[2].Tempo := S5T#1S;
   TimeWeldingPP18[3].Tempo := S5T#1S;
   TimeWeldingPP18[4].Tempo := S5T#1S;
   TimeWeldingPP18[5].Tempo := S5T#1S;
   TimeWeldingPP18[6].Tempo := S5T#1S;
   TimeWeldingPP18[7].Tempo := S5T#1S;
   TimeWeldingPP18[8].Tempo := S5T#1S;
   TimeWeldingPP18[9].Tempo := S5T#1S;
   TimeWeldingPP18[10].Tempo := S5T#1S;
   TimeWeldingPP18[11].Tempo := S5T#1S;
   TimeWeldingPP18[12].Tempo := S5T#1S;
   TimeWeldingPP18[13].Tempo := S5T#1S;
   TimeWeldingPP18[14].Tempo := S5T#1S;
   TimeWeldingPP18[15].Tempo := S5T#1S;
   TimeWeldingPP18[16].Tempo := S5T#1S;
   TimeWeldingPP18[17].Tempo := S5T#1S;
   TimeWeldingPP18[18].Tempo := S5T#1S;
   TimeWeldingPP18[19].Tempo := S5T#1S;
   TimeWeldingPP18[20].Tempo := S5T#1S;
   TimeWeldingPP19[1].Tempo := S5T#1S;
   TimeWeldingPP19[2].Tempo := S5T#1S;
   TimeWeldingPP19[3].Tempo := S5T#1S;
   TimeWeldingPP19[4].Tempo := S5T#1S;
   TimeWeldingPP19[5].Tempo := S5T#1S;
   TimeWeldingPP19[6].Tempo := S5T#1S;
   TimeWeldingPP19[7].Tempo := S5T#1S;
   TimeWeldingPP19[8].Tempo := S5T#1S;
   TimeWeldingPP19[9].Tempo := S5T#1S;
   TimeWeldingPP19[10].Tempo := S5T#1S;
   TimeWeldingPP19[11].Tempo := S5T#1S;
   TimeWeldingPP19[12].Tempo := S5T#1S;
   TimeWeldingPP19[13].Tempo := S5T#1S;
   TimeWeldingPP19[14].Tempo := S5T#1S;
   TimeWeldingPP19[15].Tempo := S5T#1S;
   TimeWeldingPP19[16].Tempo := S5T#1S;
   TimeWeldingPP19[17].Tempo := S5T#1S;
   TimeWeldingPP19[18].Tempo := S5T#1S;
   TimeWeldingPP19[19].Tempo := S5T#1S;
   TimeWeldingPP19[20].Tempo := S5T#1S;
   TimeWeldingPP20[1].Tempo := S5T#1S;
   TimeWeldingPP20[2].Tempo := S5T#1S;
   TimeWeldingPP20[3].Tempo := S5T#1S;
   TimeWeldingPP20[4].Tempo := S5T#1S;
   TimeWeldingPP20[5].Tempo := S5T#1S;
   TimeWeldingPP20[6].Tempo := S5T#1S;
   TimeWeldingPP20[7].Tempo := S5T#1S;
   TimeWeldingPP20[8].Tempo := S5T#1S;
   TimeWeldingPP20[9].Tempo := S5T#1S;
   TimeWeldingPP20[10].Tempo := S5T#1S;
   TimeWeldingPP20[11].Tempo := S5T#1S;
   TimeWeldingPP20[12].Tempo := S5T#1S;
   TimeWeldingPP20[13].Tempo := S5T#1S;
   TimeWeldingPP20[14].Tempo := S5T#1S;
   TimeWeldingPP20[15].Tempo := S5T#1S;
   TimeWeldingPP20[16].Tempo := S5T#1S;
   TimeWeldingPP20[17].Tempo := S5T#1S;
   TimeWeldingPP20[18].Tempo := S5T#1S;
   TimeWeldingPP20[19].Tempo := S5T#1S;
   TimeWeldingPP20[20].Tempo := S5T#1S;
END_DATA_BLOCK

DATA_BLOCK "DB180"	// DB 180
VERSION : 0.1
"FB24 - Gestione Mov Assi"
BEGIN
END_DATA_BLOCK

DATA_BLOCK "DB181"	// DB 181
VERSION : 0.1
"FB24 - Gestione Mov Assi"
BEGIN
END_DATA_BLOCK

ORGANIZATION_BLOCK "MAIN PROGRAM"	// OB 1
TITLE = "Main Program Sweep (Cycle)"
VERSION : 0.1
VAR_TEMP
  OB1_EV_CLASS : BYTE ;	//Bits 0-3 = 1 (Coming event), Bits 4-7 = 1 (Event class 1)
  OB1_SCAN_1 : BYTE ;	//1 (Cold restart scan 1 of OB 1), 3 (Scan 2-n of OB 1)
  OB1_PRIORITY : BYTE ;	//Priority of OB Execution
  OB1_OB_NUMBR : BYTE ;	//1 (Organization block 1, OB1)
  OB1_RESERVED_1 : BYTE ;	//Reserved for system
  OB1_RESERVED_2 : BYTE ;	//Reserved for system
  OB1_PREV_CYCLE : INT ;	//Cycle time of previous OB1 scan (milliseconds)
  OB1_MIN_CYCLE : INT ;	//Minimum cycle time of OB1 (milliseconds)
  OB1_MAX_CYCLE : INT ;	//Maximum cycle time of OB1 (milliseconds)
  OB1_DATE_TIME : DATE_AND_TIME ;	//Date and time OB1 started
END_VAR
BEGIN
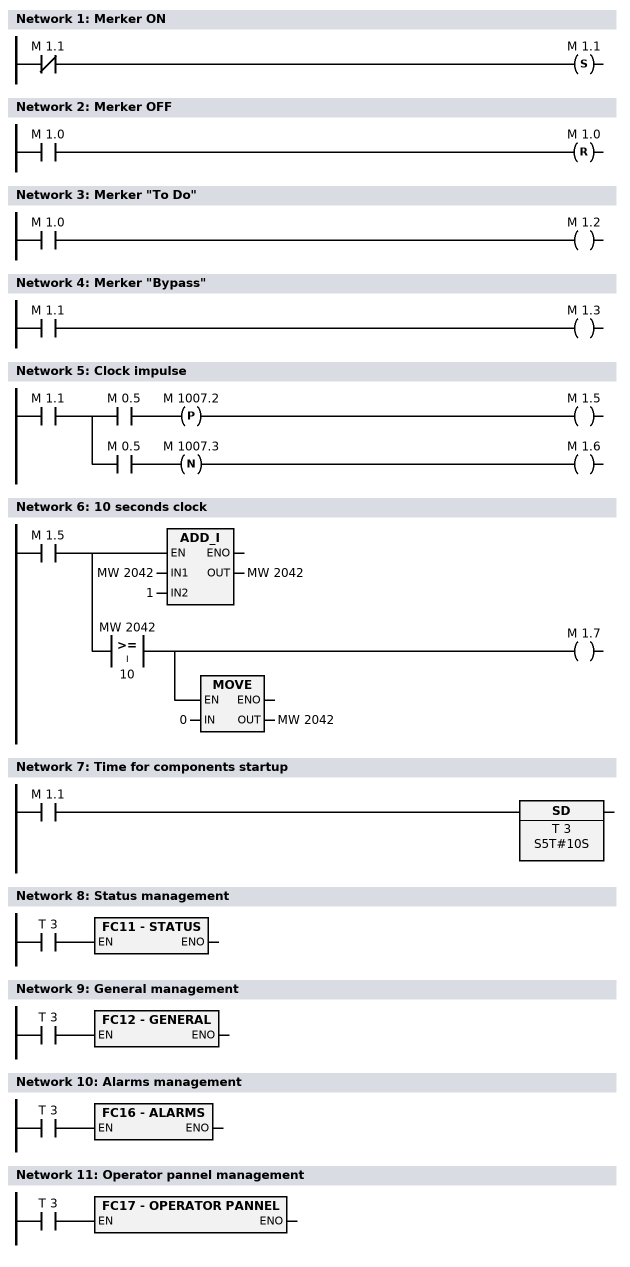
NETWORK
TITLE = Merker ON
      AN    M 1.1;
      S     M 1.1;
NETWORK
TITLE = Merker OFF
      A     M 1.0;
      R     M 1.0;
NETWORK
TITLE = Merker "To Do"
      A     M 1.0;
      =     M 1.2;
NETWORK
TITLE = Merker "Bypass"
      A     M 1.1;
      =     M 1.3;
NETWORK
TITLE = Clock impulse
      A     M 1.1;
      =     L 20.0;
      A     L 20.0;
      A     M 0.5;
      FP    M 1007.2;
      =     M 1.5;
      A     L 20.0;
      A     M 0.5;
      FN    M 1007.3;
      =     M 1.6;
NETWORK
TITLE = 10 seconds clock
      A     M 1.5;
      =     L 20.0;
      A     L 20.0;
      JNB   _001;
      L     MW 2042;
      L     1;
      +I;
      T     MW 2042;
_001: NOP   0;
      A     L 20.0;
      A(;
      L     MW 2042;
      L     10;
      >=I;
      );
      =     L 20.1;
      A     L 20.1;
      BLD   102;
      =     M 1.7;
      A     L 20.1;
      JNB   _002;
      L     0;
      T     MW 2042;
_002: NOP   0;
NETWORK
TITLE = Time for components startup
      A     M 1.1;
      L     S5T#10S;
      SD    T 3;
NETWORK
TITLE = Status management
      A     T 3;
      JNB   _003;
      CALL  "FC11 - STATUS";
_003: NOP   0;
NETWORK
TITLE = General management
      A     T 3;
      JNB   _004;
      CALL  "FC12 - GENERAL";
_004: NOP   0;
NETWORK
TITLE = Alarms management
      A     T 3;
      JNB   _005;
      CALL  "FC16 - ALARMS";
_005: NOP   0;
NETWORK
TITLE = Operator pannel management
      A     T 3;
      JNB   _006;
      CALL  "FC17 - OPERATOR PANNEL";
_006: NOP   0;
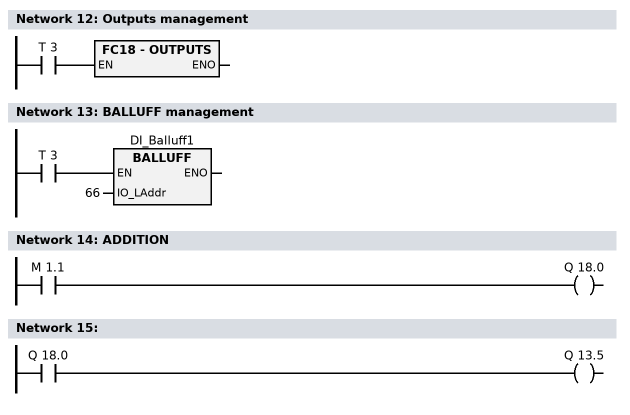
NETWORK
TITLE = Outputs management
      A     T 3;
      JNB   _007;
      CALL  "FC18 - OUTPUTS";
_007: NOP   0;
NETWORK
TITLE = BALLUFF management
      A     T 3;
      JNB   _008;
      CALL  "BALLUFF" , "DI_Balluff1" (
           IO_LAddr                 := 66);
_008: NOP   0;
NETWORK
TITLE = ADDITION
      A     M 1.1;
      =     Q 18.0;
NETWORK
TITLE =
      A     Q 18.0;
      =     Q 13.5;
END_ORGANIZATION_BLOCK

ORGANIZATION_BLOCK "I/O_FLT1"	// OB 82
TITLE = "I/O Point Fault"
VERSION : 1.0
VAR_TEMP
  OB82_EV_CLASS : BYTE ;	// 16#39, Event class 3, entering event state, internal fault event
  OB82_FLT_ID : BYTE ;	// 16#XX, Fault identification code
  OB82_PRIORITY : BYTE ;	// 26/28 (Priority of 1 is lowest)
  OB82_OB_NUMBR : BYTE ;	// 82 (Organization block 82, OB82)
  OB82_RESERVED_1 : BYTE ;	// Reserved for system
  OB82_IO_FLAG : BYTE ;	// Input (01010100), Output (01010101)
  OB82_MDL_ADDR : INT ;	// Base address of module with fault
  OB82_MDL_DEFECT : BOOL ;	// Module defective
  OB82_INT_FAULT : BOOL ;	// Internal fault
  OB82_EXT_FAULT : BOOL ;	// External fault
  OB82_PNT_INFO : BOOL ;	// Point information
  OB82_EXT_VOLTAGE : BOOL ;	// External voltage low
  OB82_FLD_CONNCTR : BOOL ;	// Field wiring connector missing
  OB82_NO_CONFIG : BOOL ;	// Module has no configuration data
  OB82_CONFIG_ERR : BOOL ;	// Module has configuration error
  OB82_MDL_TYPE : BYTE ;	// Type of module
  OB82_SUB_NDL_ERR : BOOL ;	// Sub-Module is missing or has error
  OB82_COMM_FAULT : BOOL ;	// Communication fault
  OB82_MDL_STOP : BOOL ;	// Module is stopped
  OB82_WTCH_DOG_FLT : BOOL ;	// Watch dog timer stopped module
  OB82_INT_PS_FLT : BOOL ;	// Internal power supply fault
  OB82_PRIM_BATT_FLT : BOOL ;	// Primary battery is faulty
  OB82_BCKUP_BATT_FLT : BOOL ;	// Backup battery is faulty
  OB82_RESERVED_2 : BOOL ;	// Reserved for system
  OB82_RACK_FLT : BOOL ;	// Rack fault, only for bus interface module
  OB82_PROC_FLT : BOOL ;	// Processor fault
  OB82_EPROM_FLT : BOOL ;	// EPROM fault
  OB82_RAM_FLT : BOOL ;	// RAM fault
  OB82_ADU_FLT : BOOL ;	// ADC fault
  OB82_FUSE_FLT : BOOL ;	// Fuse fault
  OB82_HW_INTR_FLT : BOOL ;	// Hardware interrupt input faulty
  OB82_RESERVED_3 : BOOL ;	// Reserved for system
  OB82_DATE_TIME : DATE_AND_TIME ;	// Date and time OB82 started
END_VAR
BEGIN
NETWORK
TITLE =
END_ORGANIZATION_BLOCK

ORGANIZATION_BLOCK "RACK_FLT"	// OB 86
TITLE = "Loss Of Rack Fault"
VERSION : 0.1
VAR_TEMP
  OB86_EV_CLASS : BYTE ;	//16#38/39 Event class 3
  OB86_FLT_ID : BYTE ;	//16#C1/C4/C5, Fault identifcation code
  OB86_PRIORITY : BYTE ;	//Priority of OB Execution
  OB86_OB_NUMBR : BYTE ;	//86 (Organization block 86, OB86)
  OB86_RESERVED_1 : BYTE ;	//Reserved for system
  OB86_RESERVED_2 : BYTE ;	//Reserved for system
  OB86_MDL_ADDR : WORD ;	//Base address of IM module in rack with fault
  OB86_RACKS_FLTD : ARRAY  [0 .. 31 ] OF BOOL ;	//Racks in fault
  OB86_DATE_TIME : DATE_AND_TIME ;	//Date and time OB86 started
END_VAR
BEGIN
NETWORK
TITLE =
END_ORGANIZATION_BLOCK

ORGANIZATION_BLOCK "COMPLETE RESTART"	// OB 100
TITLE = "Complete Restart"
VERSION : 0.1
VAR_TEMP
  OB100_EV_CLASS : BYTE ;	//16#13, Event class 1, Entering event state, Event logged in diagnostic buffer
  OB100_STRTUP : BYTE ;	//16#81/82/83/84 Method of startup
  OB100_PRIORITY : BYTE ;	//Priority of OB Execution
  OB100_OB_NUMBR : BYTE ;	//100 (Organization block 100, OB100)
  OB100_RESERVED_1 : BYTE ;	//Reserved for system
  OB100_RESERVED_2 : BYTE ;	//Reserved for system
  OB100_STOP : WORD ;	//Event that caused CPU to stop (16#4xxx)
  OB100_STRT_INFO : DWORD ;	//Information on how system started
  OB100_DATE_TIME : DATE_AND_TIME ;	//Date and time OB100 started
END_VAR
BEGIN
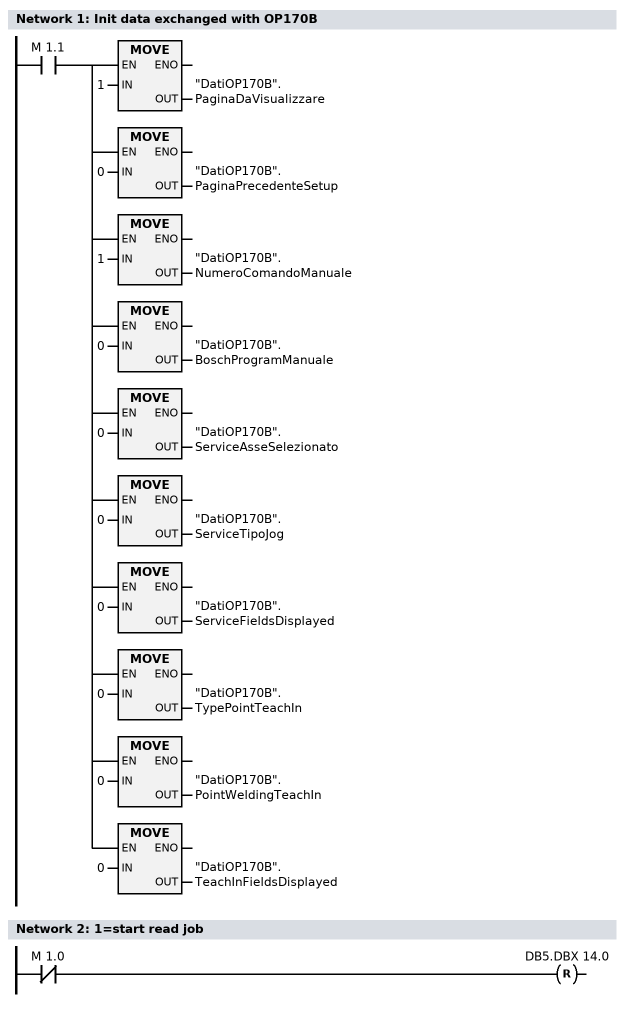
NETWORK
TITLE = Init data exchanged with OP170B
      A     M 1.1;
      =     L 20.0;
      A     L 20.0;
      JNB   _001;
      L     1;
      T     "DatiOP170B".PaginaDaVisualizzare;
_001: NOP   0;
      A     L 20.0;
      JNB   _002;
      L     0;
      T     "DatiOP170B".PaginaPrecedenteSetup;
_002: NOP   0;
      A     L 20.0;
      JNB   _003;
      L     1;
      T     "DatiOP170B".NumeroComandoManuale;
_003: NOP   0;
      A     L 20.0;
      JNB   _004;
      L     0;
      T     "DatiOP170B".BoschProgramManuale;
_004: NOP   0;
      A     L 20.0;
      JNB   _005;
      L     0;
      T     "DatiOP170B".ServiceAsseSelezionato;
_005: NOP   0;
      A     L 20.0;
      JNB   _006;
      L     0;
      T     "DatiOP170B".ServiceTipoJog;
_006: NOP   0;
      A     L 20.0;
      JNB   _007;
      L     0;
      T     "DatiOP170B".ServiceFieldsDisplayed;
_007: NOP   0;
      A     L 20.0;
      JNB   _008;
      L     0;
      T     "DatiOP170B".TypePointTeachIn;
_008: NOP   0;
      A     L 20.0;
      JNB   _009;
      L     0;
      T     "DatiOP170B".PointWeldingTeachIn;
_009: NOP   0;
      A     L 20.0;
      JNB   _00a;
      L     0;
      T     "DatiOP170B".TeachInFieldsDisplayed;
_00a: NOP   0;
NETWORK
TITLE = 1=start read job
      AN    M 1.0;
      R     DB5.DBX 14.0;
END_ORGANIZATION_BLOCK

ORGANIZATION_BLOCK "MOD_ERR"	// OB 122
TITLE = "Module Access Error"
VERSION : 0.1
VAR_TEMP
  OB122_EV_CLASS : BYTE ;	//16#29, Event class 2, Entering event state, Internal fault event
  OB122_SW_FLT : BYTE ;	//16#XX Software error code
  OB122_PRIORITY : BYTE ;	//Priority of OB Execution
  OB122_OB_NUMBR : BYTE ;	//122 (Organization block 122, OB122)
  OB122_BLK_TYPE : BYTE ;	//16#88/8C/8E Type of block fault occured in
  OB122_MEM_AREA : BYTE ;	//Memory area where access error occured
  OB122_MEM_ADDR : WORD ;	//Memory address where access error occured
  OB122_BLK_NUM : WORD ;	//Block number in which error occured
  OB122_PRG_ADDR : WORD ;	//Program address where error occured
  OB122_DATE_TIME : DATE_AND_TIME ;	//Date and time OB1 started
END_VAR
BEGIN
NETWORK
TITLE =
END_ORGANIZATION_BLOCK
